// TIA Portal V20 export
TYPE "LER_typeBrakeTestEmInterface"
// stored: Access Published
   STRUCT
      commands : "LER_typeBrakeTestEmHmiCommands";
      monitoring { ExternalWritable := 'False'} : "LER_typeBrakeTestEmMonitoring";
   END_STRUCT;
END_TYPE
